HMI tags "03.PumpControl"
   "Stop" : Bool AT %M0.1, T100ms
   "Lo" : Bool AT %M0.2, T100ms
   "Start" : Bool AT %M0.0, T100ms
   "Hi" : Bool AT %M0.3, T100ms
   "P_1" : Bool AT %M0.4, T100ms
   "P_2" : Bool AT %M0.5, T100ms
   "P_3" : Bool AT %M0.6, T100ms
   "L" : Int AT %MW4, T100ms

text list "SystemTextList_ConfigErrorAlarmTextLibrary_1": 1 'NameService configuration error: Implicit deletion. Subelement instance @6%s@ must be deleted explicitly.'; 2 'NameService configuration error: Implicit deletion. Alias/Format/Unit instance @6%s@ must be deleted explicitly.'

text list "SystemTextList_ConfigErrorAlarmTextLibrary_2": 1 'EvDpManager::cleanupDeletedDatapoint - alert handler config is deleted implicitly for deleted datapoint, @3%s@'; 2 'EvDpManager::cleanupDeletedDatapoint - alert handler config is deleted implicitly but still has overrides, @3%s@'; 3 'EvDpManager::cleanupDeletedDatapoint - default value config is deleted implicitly for deleted datapoint, @3%s@'; 4 'EvDpManager::cleanupDeletedDatapoint - default value config is deleted implicitly but still has overrides, @3%s@'; 5 'EvDpManager::cleanupDeletedDatapoint - initial value config is deleted implicitly for deleted datapoint, @3%s@'; 6 'EvDpManager::cleanupDeletedDatapoint - initial value config is deleted implicitly but still has overrides, @3%s@'; 7 'EvDpManager::cleanupDeletedDatapoint - distribution config is deleted implicitly for deleted datapoint, @3%s@'; 8 'EvDpManager::cleanupDeletedDatapoint - distribution config is deleted implicitly but still has overrides, @3%s@'; 9 'EvDpManager::cleanupDeletedDatapoint - rangeCheck config is deleted implicitly for deleted datapoint, @3%s@'; 10 'EvDpManager::cleanupDeletedDatapoint - rangeCheck config is deleted implicitly but still has overrides, @3%s@'

text list "SystemTextList_ConfigErrorAlarmTextLibrary_3": 1 'The configured data point type was deleted, but a configured type is still defined for the node type: @3%s@.'; 2 'The configured data point node type was deleted in the data point type, but a configured type is still defined for the element: @3%s@.'

text list "SystemTextList_ConfigErrorAlarmTextLibrary_4": 2 'Cycles: @6%s@ does not exist'; 3 'Alarms: @6%s@ exists already'; 4 'Tags: Address @6%s@ was rejected'; 1 'Connections: @6%s@ does not exist'; 5 'Tags: Acquisition mode @6%s@ is not supported.'; 6 'Cycles: @6%s@ was deleted but associated tags exist.'; 7 'Connections: @6%s@ was deleted but associated tags exist.'; 8 'Tags: Tag @6%s@ was rejected.'; 9 'Tags: Tag @6%s@ has an invalid value.'; 0 'Connections: Connection to @6%s@ could not be established.'; 65638 'Connections: Connection to @6%s@ could not be established.'; 65639 'Connections: @6%s@ disconnected.'; 65640 'Connections: Connection to the HMI device @6%s@ is lost.'; 65641 'Connections: Connection to the PLC @6%s@ is lost.'; 65541 'Connections: Timeout while establishing the connection to @6%s@.'; 65542 'Connections: @6%s@ faulty.'; 65543 'Connections: Connection to the HMI device disconnected. Connection @5%s@ was changed.'; 65544 'Connections: Connection to the HMI device disconnected. Driver property was changed for connection @5%s@.'

text list "SystemTextList_ConfigErrorAlarmTextLibrary_5": 1 'Connections: Lifecycle monitoring cycle must be shorter than the response time.'; 2 'Connections: Cyclic services are configured but not supported by the target device.'; 3 'Connections: Change-controlled reading is configured but not supported by the target device.'; 4 'Tags: The address @6%s@ does not exist in the PLC.'; 5 'Tags: The default conversion type for the address @6%s@ could not be determined.'; 6 'Tags: Invalid conversion type'; 7 'Cycles: Invalid conversion type. Conversion is not supported at HmiCycle.'; 4096 'Connections: Version of the address @6%s@ is not supported.'; 4097 'Connections: PROFIBUS address is not supported.'; 4098 'Connections: Softbus address is not supported.'; 4099 'Connections: Address type @6%s@ is not supported.'; 4100 'Connections: Invalid connection name @6%s@. Access point is being ignored.'; 4101 'Connections: Routing is not supported. @6%s@ is not used.'; 4102 'Connections: Routing is not supported. @6%s@ is not used.'; 4103 'Connections: Invalid IP address @6%s@'; 4104 'Connections: Invalid Named Connection @6%s@. Valid format: >VMD</>connection<'; 4105 'Connections: Invalid Named Connection @6%s@. VMD connection name is too long. Only 24 characters are permitted.'; 4106 'Connections: Invalid Named Connection @6%s@. Connection name is too long. Only 32 characters are permitted.'; 4107 'Connections: Rack number @6%s@ is outside of the permitted range (0..7)'; 4108 'Connections: Invalid Named Connection @6%s@. Rack is ignored.'; 4109 'Connections: Slot number @6%s@ is outside of the permitted range (0..31)'; 4110 'Connections: Invalid Named Connection @6%s@. Slot is ignored.'; 4111 'Connection could not be established. Maximum number of available connections (@6%s@) has been exceeded.'; 4112 'Connection aborted. No sign of life in the last @4%s@ ms.'; 4113 'Connection could not be established - @4%s@'; 4114 'Connection could not be established. The address @6%s@ cannot be used.'; 4115 'Connection could not be established. Invalid address @6%s@'; 4116 'Connection could not be established - @4%s@'

text list "SystemTextList_ConfigErrorAlarmTextLibrary_6": 1 'Connection could not be established. Application instance certificate is not configured.'; 2 'Connection could not be established. Server has rejected the client certificate. OPC UA status code @4%s@.'; 3 'Connection could not be established. Internal problem in the certificate store. OPC UA status code @4%s@'; 4 'Connection could not be established. Application instance certificate could not be loaded. OPC UA status code @4%s@'; 5 'Connection could not be established. Server has not provided a certificate. @4%s@'; 6 'Connection could not be established. Validation of server certificate has failed. OPC UA status code @4%s@.'; 7 'Connection was closed. Error during alarm synchronization. OPC UA status code @4%s@.'; 8 'Connection was closed. Alarm/event subscription has failed. The number of operations on the server has been exceeded.'; 9 'Connection was closed. Alarm/event subscription has failed. The number of alarm/event subscriptions on the server has been exceeded.'; 10 'Connection could not be established. Server reports a license problem. OPC UA status code @4%s@.'; 11 'Connection could not be established. Maximum number of server sessions has been exceeded.'; 12 'Connection could not be established. Safety configuration is inconsistent. @4%s@'; 13 'Connection could not be established. The address @4%s@ cannot be used.'; 14 'Connection could not be established. OPC UA status code @4%s@'; 15 'Connection aborted. OPC UA server was stopped.'; 16 'Connection aborted. No sign of life in the last @4%s@ ms.'; 17 'Connection was closed. OPC UA server maintenance.'; 18 'Connection could not be established. Invalid configuration of the authentication mode - @4%s@'; 19 'Connection could not be established. User could not be authenticated. OPC UA status code @4%s@'; 20 'Connection could not be established. Server does not permit anonymous connection. OPC UA status code @4%s@'; 21 'Connection could not be established. Certificate problem: Error when writing the safety-relevant data to @4%s@.'; 22 'Connection could not be established. Certificate problem: Unexpected file in the folder @4%s@ cannot be removed.'; 23 'Connection could not be established. User could not be authenticated. No user or password configured.'; 24 'Connection could not be established. Unexpected length of the server certificate. @4%s@'; 25 'Connection could not be established. @4%s@ is empty.'; 26 'Connection could not be established. @4%s@ has an unexpected format.'; 27 'Connection could not be established. Server endpoints cannot be read. OPC UA status code @4%s@'; 28 'Connection could not be established. No server endpoints were found. @4%s@'; 29 'Connection could not be established. Application instance certificate could not be found.'; 30 'Connection could not be established. Unexpected format of the certificate @4%s@.'; 31 'Connection could not be established. Unexpected format of the certificate block list @4%s@.'; 32 'Connection could not be established. User could not be authenticated. An encryption detail is invalid. @4%s@'; 34 'Connection could not be established. - The configured non-transparent redundancy mode @4%s@ is not supported.'; 101 'Tags: Address @6%s@ does not exist on the server.'; 103 'Tags: Address @6%s@ cannot be accessed.'; 104 'Tags: Acquisition mode is not supported for address @6%s@.'; 201 'Alarms: Address @6%s@ does not exist on the server.'; 202 'Alarms: Address @6%s@ cannot be used. The specified range filter is not an OPC UA Event Notifier.'; 203 'Alarms: Address @6%s@ cannot be used. The specified range filter does not exist on the server.'; 204 'Alarms: Address @6%s@ cannot be used because it is not an OPC UA event type.'; 205 'Alarms: Address @6%s@ cannot be used because the OPC UA condition type is not supported.'; 206 'Alarms: Address @6%s@ cannot be used because the event type does not exist on the server.'; 207 'Alarms: Acquisition type cannot be used for address @6%s@.'; 301 'Address @6%s@ cannot be used because the version number is missing.'; 302 'Address @6%s@ cannot be used because the version number is invalid.'; 303 'Address @6%s@ cannot be used because the number of '$' delimiters is invalid.'; 304 'Address @6%s@ cannot be used because the address type is invalid.'; 305 'Unsupported version @6%s@ of the address'; 401 'Unexpected OPC UA server response: @6%s@'

text list "SystemTextList_ConfigErrorAlarmTextLibrary_7": 1 'Messages: Invalid condition string for the alarm view @6%s@.'; 2 'Messages: Invalid status tag and bit for the alarm view @6%s@.'; 3 'Messages: Invalid control tag and bit for the alarm view @6%s@.'

text list "SystemTextList_ConfigErrorAlarmTextLibrary_8": 1 'Logs: Implicit deletion. Logging tag instance @6%s@ should be deleted but there are overloaded elements.'

text list "SystemTextList_ConfigErrorAlarmTextLibrary_9": 2 'Restart of the runtime is required.'; 3 'The correct storage medium must be ejected and inserted again.'

text list "SystemTextList_ConfigErrorAlarmTextLibrary_10": 1 'CDS cache - Cache folder cannot be created or reached: @6%s@'; 2 'LOC cache - Cache folder cannot be created or reached: @6%s@'

text list "SystemTextList_ConfigErrorAlarmTextLibrary_11": 2 'and synchronization will start automatically. Shutting down either of them during synchronization will not cause data loss.'; 3 'and synchronization is scheduled for: @5%Y-%m-%d %H:%M:%S@. Shutting down either of the computers will not cause data loss.'

text list "SystemTextList_RuntimeCollaborationFailureReason_1": 0 'Unknown error (@3%s@)'; 1 'The system is not running or there is a network problem'; 2 'Runtime is not started on the target device.'; 3 'The System ID does not match the expected System ID (@3%s@)'; 4 'The Collaboration name does not match the expected Collaboration name '@3%s@''; 5 'Wrong or unknown certificate'; 6 'Revoked certificate'; 7 'The time difference is too big.'; 8 'No common supported message version'; 9 'System ID (@3%s@) already exists'; 10 'System name (@3%s@) already exists'; 11 'ID/Name in local configuration for Runtime Collaboration already exists'

text list "SystemTextList_RedundancyRecoveryFailureReason_1": 0 'Data recovery request temporarily rejected until own recovery request has been responded to.'; 1 'Data recovery request rejected. Online backup running.'; 2 'Data recovery request rejected. Connection to the Event Manager is not established.'; 3 'Data recovery request temporarily rejected until delta activation is complete.'; 4 'Data recovery request temporarily rejected until alarms and tags are retentive.'; 5 'Data recovery request rejected. The obligatory file config.level.es is missing on the computer.'; 6 'Data recovery request was canceled by the Event Manager.'; 7 'The data synchronization between the devices has failed.'

text list "SystemTextList_S7PlusAlarmTextListCollection_1": 4096 'Connections: Connection to the PLC @4%s@ is lost'; 4097 'Connections: Connection to the HMI device @4%s@ is lost'; 4098 'Connections: Maximum number of connections exceeded - @4%s@'; 4099 'Out of resources on PLC - @4%s@'; 4100 'Legitimation failed, invalid or missing password - @4%s@'; 4101 'Request to open the connection failed - @4%s@'; 4102 'Connections: Cannot connect to PLC - @4%s@'; 4103 'Request to open the connection could not be sent'; 4104 'General certificate error for PLC - @4%s@'; 4105 'PLC certificate expired for PLC - @4%s@'; 4106 'PLC certificate is revoked for PLC - @4%s@'; 4107 'PLC certificate is untrustworthy. Manual trust is possible for - @4%s@'; 4108 'PLC certificate is untrustworthy. Manual trust is not possible for - @4%s@'

text list "SystemTextList_AllenBradleyEIPAlarmTextListCollection_7": 4096 'Connection lost on PLC side - @5%s@'; 4097 'Connection lost on HMI side - @5%s@'; 4098 'Maximum number of connections exceeded - @5%s@'; 4099 'Out of resources on PLC - @5%s@'; 4100 'Legitimation failed, invalid or missing password - @5%s@'; 4101 'Open request failed - @5%s@'; 4102 'Cannot connect to PLC - @5%s@'; 4103 'Open request could not be sent'; 4104 'root certificate expired for - @5%s@'; 4105 'PLC certificate untrusted for - @5%s@'

text list "SystemTextList_AllenBradleyDF1AlarmTextListCollection_9": 4096 'Connections: Connection to the PLC @5%s@ is lost'; 4097 'Connections: Connection to the HMI device @5%s@ is lost'; 4098 'Connections: Maximum number of connections exceeded - @5%s@'; 4099 'Out of resources on PLC - @5%s@'; 4100 'Legitimation failed, invalid or missing password - @5%s@'; 4101 'Request to open the connection failed - @5%s@'; 4102 'Connections: Cannot connect to PLC - @5%s@'; 4103 'Request to open the connection could not be sent'; 4104 'General certificate error for PLC - @5%s@'; 4105 'PLC certificate expired for PLC - @5%s@'; 4106 'PLC certificate is revoked for PLC - @5%s@'; 4107 'PLC certificate is untrustworthy. Manual trust is possible for - @5%s@'; 4108 'PLC certificate is untrustworthy. Manual trust is not possible for - @5%s@'

text list "SystemTextList_OmronEIPAlarmTextListCollection_6": 4096 'Connection lost on PLC side - @5%s@'; 4097 'Connection lost on HMI side - @5%s@'; 4098 'Maximum number of connections exceeded - @5%s@'; 4099 'Out of resources on PLC - @5%s@'; 4100 'Legitimation failed, invalid or missing password - @5%s@'; 4101 'Open request failed - @5%s@'; 4102 'Cannot connect to PLC - @5%s@'; 4103 'Open request could not be sent'; 4104 'root certificate expired for - @5%s@'; 4105 'PLC certificate untrusted for - @5%s@'

text list "SystemTextList_StdModbusTCPAlarmTextListCollection_5": 4096 'Connections: Connection to the PLC @5%s@ is lost'; 4097 'Connections: Connection to the HMI device @5%s@ is lost'; 4098 'Connections: Maximum number of connections exceeded - @5%s@'; 4099 'Out of resources on PLC - @5%s@'; 4100 'Legitimation failed, invalid or missing password - @5%s@'; 4101 'Request to open the connection failed - @5%s@'; 4102 'Connections: Cannot connect to PLC - @5%s@'; 4103 'Request to open the connection could not be sent'; 4104 'General certificate error for PLC - @5%s@'; 4105 'PLC certificate expired for PLC - @5%s@'; 4106 'PLC certificate is revoked for PLC - @5%s@'; 4107 'PLC certificate is untrustworthy. Manual trust is possible for - @5%s@'; 4108 'PLC certificate is untrustworthy. Manual trust is not possible for - @5%s@'

text list "SystemTextList_MitsubishiMCAlarmTextListCollection_4": 4096 'Connection lost on PLC side - @5%s@'; 4097 'Connection lost on HMI side - @5%s@'; 4098 'Maximum number of connections exceeded - @5%s@'; 4099 'Out of resources on PLC - @5%s@'; 4100 'Legitimation failed, invalid or missing password - @5%s@'; 4101 'Open request failed - @5%s@'; 4102 'Cannot connect to PLC - @5%s@'; 4103 'Open request could not be sent'; 4104 'root certificate expired for - @5%s@'; 4105 'PLC certificate untrusted for - @5%s@'

text list "SystemTextList_MitsubishiiQAlarmTextListCollection_3": 4096 'Connection lost on PLC side - @5%s@'; 4097 'Connection lost on HMI side - @5%s@'; 4098 'Maximum number of connections exceeded - @5%s@'; 4099 'Out of resources on PLC - @5%s@'; 4100 'Legitimation failed, invalid or missing password - @5%s@'; 4101 'Open request failed - @5%s@'; 4102 'Cannot connect to PLC - @5%s@'; 4103 'Open request could not be sent'; 4104 'root certificate expired for - @5%s@'; 4105 'PLC certificate untrusted for - @5%s@'

text list "SystemTextList_StdModbusRTUAlarmTextListCollection_8": 4096 'Connections: Connection to the PLC @5%s@ is lost'; 4097 'Connections: Connection to the HMI device @5%s@ is lost'; 4098 'Connections: Maximum number of connections exceeded - @5%s@'; 4099 'Out of resources on PLC - @5%s@'; 4100 'Legitimation failed, invalid or missing password - @5%s@'; 4101 'Request to open the connection failed - @5%s@'; 4102 'Connections: Cannot connect to PLC - @5%s@'; 4103 'Request to open the connection could not be sent'; 4104 'General certificate error for PLC - @5%s@'; 4105 'PLC certificate expired for PLC - @5%s@'; 4106 'PLC certificate is revoked for PLC - @5%s@'; 4107 'PLC certificate is untrustworthy. Manual trust is possible for - @5%s@'; 4108 'PLC certificate is untrustworthy. Manual trust is not possible for - @5%s@'

text list "SystemTextList_LogoAlarmTextListCollection_10": 4096 'Connections: Connection to the PLC @5%s@ is lost'; 4097 'Connections: Connection to the HMI device @5%s@ is lost'; 4098 'Connections: Maximum number of connections exceeded - @5%s@'; 4099 'Out of resources on PLC - @5%s@'; 4100 'Legitimation failed, invalid or missing password - @5%s@'; 4101 'Request to open the connection failed - @5%s@'; 4102 'Connections: Cannot connect to PLC - @5%s@'; 4103 'Request to open the connection could not be sent'; 4104 'General certificate error for PLC - @5%s@'; 4105 'PLC certificate expired for PLC - @5%s@'; 4106 'PLC certificate is revoked for PLC - @5%s@'; 4107 'PLC certificate is untrustworthy. Manual trust is possible for - @5%s@'; 4108 'PLC certificate is untrustworthy. Manual trust is not possible for - @5%s@'

graphic list "Switch": 0 'rotary-switches-open'; 1 'rotary-switches-close'

graphic list "Light": 0 'light_green_off'; 1 'light_green_on'

graphic list "Agitator": 0 'agitator_1'; 1 'agitator_2'; 2 'agitator_3'; 3 'agitator_4'
*)

(* ===== HMI "HiddenHmiRTDeviceFaceplateTypes" =====

HMI tags "0daced1d-1c12-4c0f-a1c7-efedc7fbd37d"
   "Data" : f64981b7-23c1-4b9c-90a3-7c9aa74d9c52, internal
*)

(* ===== HMI "HiddenHmiRTDeviceFaceplateTypes" =====

HMI tags "0daced1d-1c12-4c0f-a1c7-efedc7fbd37d"
   "Data" : f64981b7-23c1-4b9c-90a3-7c9aa74d9c52, internal
*)

(* ===== HMI "HMI_RT_4" =====
connection "UA_Connection_1": SCADA_OPC, ILRT_OPC_UA
connection "S7_Connection_1": ETHERNET, ILRT_S7_1500_OMS

HMI tags "01.HeaterONOFFCtrl"
   "Temp_SP" : Float AT ns=http://www.siemens.com/simatic-s7-opcua;s="ON_OFF_Ctrl_1"."SP", T100ms
   "Temp" : Float AT ns=http://www.siemens.com/simatic-s7-opcua;s="ON_OFF_Ctrl_1"."T", T100ms
   "Enable" : Boolean AT ns=http://www.siemens.com/simatic-s7-opcua;s="ON_OFF_Ctrl_1"."Enable", T100ms
   "Ready" : Boolean AT ns=http://www.siemens.com/simatic-s7-opcua;s="HeaterSim_1"."Ready", T100ms
   "Fault" : Boolean AT ns=http://www.siemens.com/simatic-s7-opcua;s="HeaterSim_1"."Fault", T100ms

HMI tags "02.MotorDOLCtrl"
   "Theta" : Float AT ns=http://www.siemens.com/simatic-s7-opcua;s="MotorSim_1"."Theta", T100ms
   "Omega" : Real AT %DB4.DBD8, T100ms
   "EnableCtrl" : Boolean AT ns=http://www.siemens.com/simatic-s7-opcua;s="DOL_Ctrl_1"."Enable", T100ms
   "i_set" : Float AT ns=http://www.siemens.com/simatic-s7-opcua;s="DOL_Ctrl_1"."i_set", T100ms
   "RunCmd" : Boolean AT ns=http://www.siemens.com/simatic-s7-opcua;s="DOL_Ctrl_1"."RunCmd", T100ms
   "MotorFault" : Boolean AT ns=http://www.siemens.com/simatic-s7-opcua;s="MotorSim_1"."Fault", T100ms
   "MotorReady" : Boolean AT ns=http://www.siemens.com/simatic-s7-opcua;s="MotorSim_1"."Ready", T100ms

HMI tags "03.HeaterPIDCtrl"
   "Temperature_SP" : Real AT %DB6.DBD2, T100ms
   "Temperature" : Real AT %DB7.DBD8, T100ms
   "EnableHeaterCtrl" : Bool AT %DB6.DBX0.0, T100ms
   "HeaterReady" : Bool AT %DB7.DBX12.0, T100ms
   "Kp" : Real AT %DB6.DBD12, T100ms
   "Ki" : Real AT %DB6.DBD16, T100ms
   "Kd" : Real AT %DB6.DBD20, T100ms
   "u" : Real AT %DB6.DBD32, T100ms

HMI tags "04.MotorPIDCtrl"
   "Omega_SP_Motor" : Real AT %DB10.DBD2, T100ms
   "EnablePID_Motor" : Bool AT %DB10.DBX0.0, T100ms
   "RunCmd_Motor" : Bool AT %DB9.DBX0.1, T100ms
   "Ready_Motor" : Bool AT %DB8.DBX16.0, T100ms
   "Omega_Motor" : Real AT %DB10.DBD6, T100ms
   "Kd_Motor" : Real AT %DB10.DBD10, T100ms
   "Ki_Motor" : Real AT %DB10.DBD16, T100ms
   "Kp_Motor" : Real AT %DB10.DBD20, T100ms
   "u_Motor" : Real AT %DB10.DBD32, T100ms

text list "SystemTextList_ConfigErrorAlarmTextLibrary_1": 1 'NameService configuration error: Implicit deletion. Subelement instance @6%s@ must be deleted explicitly.'; 2 'NameService configuration error: Implicit deletion. Alias/Format/Unit instance @6%s@ must be deleted explicitly.'

text list "SystemTextList_ConfigErrorAlarmTextLibrary_2": 1 'EvDpManager::cleanupDeletedDatapoint - alert handler config is deleted implicitly for deleted datapoint, @3%s@'; 2 'EvDpManager::cleanupDeletedDatapoint - alert handler config is deleted implicitly but still has overrides, @3%s@'; 3 'EvDpManager::cleanupDeletedDatapoint - default value config is deleted implicitly for deleted datapoint, @3%s@'; 4 'EvDpManager::cleanupDeletedDatapoint - default value config is deleted implicitly but still has overrides, @3%s@'; 5 'EvDpManager::cleanupDeletedDatapoint - initial value config is deleted implicitly for deleted datapoint, @3%s@'; 6 'EvDpManager::cleanupDeletedDatapoint - initial value config is deleted implicitly but still has overrides, @3%s@'; 7 'EvDpManager::cleanupDeletedDatapoint - distribution config is deleted implicitly for deleted datapoint, @3%s@'; 8 'EvDpManager::cleanupDeletedDatapoint - distribution config is deleted implicitly but still has overrides, @3%s@'; 9 'EvDpManager::cleanupDeletedDatapoint - rangeCheck config is deleted implicitly for deleted datapoint, @3%s@'; 10 'EvDpManager::cleanupDeletedDatapoint - rangeCheck config is deleted implicitly but still has overrides, @3%s@'

text list "SystemTextList_ConfigErrorAlarmTextLibrary_3": 1 'The configured data point type was deleted, but a configured type is still defined for the node type: @3%s@.'; 2 'The configured data point node type was deleted in the data point type, but a configured type is still defined for the element: @3%s@.'

text list "SystemTextList_ConfigErrorAlarmTextLibrary_4": 2 'Cycles: @6%s@ does not exist'; 3 'Alarms: @6%s@ exists already'; 4 'Tags: Address @6%s@ was rejected'; 1 'Connections: @6%s@ does not exist'; 5 'Tags: Acquisition mode @6%s@ is not supported.'; 6 'Cycles: @6%s@ was deleted but associated tags exist.'; 7 'Connections: @6%s@ was deleted but associated tags exist.'; 8 'Tags: Tag @6%s@ was rejected.'; 9 'Tags: Tag @6%s@ has an invalid value.'; 0 'Connections: Connection to @6%s@ could not be established.'; 65638 'Connections: Connection to @6%s@ could not be established.'; 65639 'Connections: @6%s@ disconnected.'; 65640 'Connections: Connection to the HMI device @6%s@ is lost.'; 65641 'Connections: Connection to the PLC @6%s@ is lost.'; 65541 'Connections: Timeout while establishing the connection to @6%s@.'; 65542 'Connections: @6%s@ faulty.'; 65543 'Connections: Connection to the HMI device disconnected. Connection @5%s@ was changed.'; 65544 'Connections: Connection to the HMI device disconnected. Driver property was changed for connection @5%s@.'

text list "SystemTextList_ConfigErrorAlarmTextLibrary_5": 1 'Connections: Lifecycle monitoring cycle must be shorter than the response time.'; 2 'Connections: Cyclic services are configured but not supported by the target device.'; 3 'Connections: Change-controlled reading is configured but not supported by the target device.'; 4 'Tags: The address @6%s@ does not exist in the PLC.'; 5 'Tags: The default conversion type for the address @6%s@ could not be determined.'; 6 'Tags: Invalid conversion type'; 7 'Cycles: Invalid conversion type. Conversion is not supported at HmiCycle.'; 4096 'Connections: Version of the address @6%s@ is not supported.'; 4097 'Connections: PROFIBUS address is not supported.'; 4098 'Connections: Softbus address is not supported.'; 4099 'Connections: Address type @6%s@ is not supported.'; 4100 'Connections: Invalid connection name @6%s@. Access point is being ignored.'; 4101 'Connections: Routing is not supported. @6%s@ is not used.'; 4102 'Connections: Routing is not supported. @6%s@ is not used.'; 4103 'Connections: Invalid IP address @6%s@'; 4104 'Connections: Invalid Named Connection @6%s@. Valid format: >VMD</>connection<'; 4105 'Connections: Invalid Named Connection @6%s@. VMD connection name is too long. Only 24 characters are permitted.'; 4106 'Connections: Invalid Named Connection @6%s@. Connection name is too long. Only 32 characters are permitted.'; 4107 'Connections: Rack number @6%s@ is outside of the permitted range (0..7)'; 4108 'Connections: Invalid Named Connection @6%s@. Rack is ignored.'; 4109 'Connections: Slot number @6%s@ is outside of the permitted range (0..31)'; 4110 'Connections: Invalid Named Connection @6%s@. Slot is ignored.'; 4111 'Connection could not be established. Maximum number of available connections (@6%s@) has been exceeded.'; 4112 'Connection aborted. No sign of life in the last @4%s@ ms.'; 4113 'Connection could not be established - @4%s@'; 4114 'Connection could not be established. The address @6%s@ cannot be used.'; 4115 'Connection could not be established. Invalid address @6%s@'; 4116 'Connection could not be established - @4%s@'

text list "SystemTextList_ConfigErrorAlarmTextLibrary_6": 1 'Connection could not be established. Application instance certificate is not configured.'; 2 'Connection could not be established. Server has rejected the client certificate. OPC UA status code @4%s@.'; 3 'Connection could not be established. Internal problem in the certificate store. OPC UA status code @4%s@'; 4 'Connection could not be established. Application instance certificate could not be loaded. OPC UA status code @4%s@'; 5 'Connection could not be established. Server has not provided a certificate. @4%s@'; 6 'Connection could not be established. Validation of server certificate has failed. OPC UA status code @4%s@.'; 7 'Connection was closed. Error during alarm synchronization. OPC UA status code @4%s@.'; 8 'Connection was closed. Alarm/event subscription has failed. The number of operations on the server has been exceeded.'; 9 'Connection was closed. Alarm/event subscription has failed. The number of alarm/event subscriptions on the server has been exceeded.'; 10 'Connection could not be established. Server reports a license problem. OPC UA status code @4%s@.'; 11 'Connection could not be established. Maximum number of server sessions has been exceeded.'; 12 'Connection could not be established. Safety configuration is inconsistent. @4%s@'; 13 'Connection could not be established. The address @4%s@ cannot be used.'; 14 'Connection could not be established. OPC UA status code @4%s@'; 15 'Connection aborted. OPC UA server was stopped.'; 16 'Connection aborted. No sign of life in the last @4%s@ ms.'; 17 'Connection was closed. OPC UA server maintenance.'; 18 'Connection could not be established. Invalid configuration of the authentication mode - @4%s@'; 19 'Connection could not be established. User could not be authenticated. OPC UA status code @4%s@'; 20 'Connection could not be established. Server does not permit anonymous connection. OPC UA status code @4%s@'; 21 'Connection could not be established. Certificate problem: Error when writing the safety-relevant data to @4%s@.'; 22 'Connection could not be established. Certificate problem: Unexpected file in the folder @4%s@ cannot be removed.'; 23 'Connection could not be established. User could not be authenticated. No user or password configured.'; 24 'Connection could not be established. Unexpected length of the server certificate. @4%s@'; 25 'Connection could not be established. @4%s@ is empty.'; 26 'Connection could not be established. @4%s@ has an unexpected format.'; 27 'Connection could not be established. Server endpoints cannot be read. OPC UA status code @4%s@'; 28 'Connection could not be established. No server endpoints were found. @4%s@'; 29 'Connection could not be established. Application instance certificate could not be found.'; 30 'Connection could not be established. Unexpected format of the certificate @4%s@.'; 31 'Connection could not be established. Unexpected format of the certificate block list @4%s@.'; 32 'Connection could not be established. User could not be authenticated. An encryption detail is invalid. @4%s@'; 34 'Connection could not be established. - The configured non-transparent redundancy mode @4%s@ is not supported.'; 101 'Tags: Address @6%s@ does not exist on the server.'; 103 'Tags: Address @6%s@ cannot be accessed.'; 104 'Tags: Acquisition mode is not supported for address @6%s@.'; 201 'Alarms: Address @6%s@ does not exist on the server.'; 202 'Alarms: Address @6%s@ cannot be used. The specified range filter is not an OPC UA Event Notifier.'; 203 'Alarms: Address @6%s@ cannot be used. The specified range filter does not exist on the server.'; 204 'Alarms: Address @6%s@ cannot be used because it is not an OPC UA event type.'; 205 'Alarms: Address @6%s@ cannot be used because the OPC UA condition type is not supported.'; 206 'Alarms: Address @6%s@ cannot be used because the event type does not exist on the server.'; 207 'Alarms: Acquisition type cannot be used for address @6%s@.'; 301 'Address @6%s@ cannot be used because the version number is missing.'; 302 'Address @6%s@ cannot be used because the version number is invalid.'; 303 'Address @6%s@ cannot be used because the number of '$' delimiters is invalid.'; 304 'Address @6%s@ cannot be used because the address type is invalid.'; 305 'Unsupported version @6%s@ of the address'; 401 'Unexpected OPC UA server response: @6%s@'

text list "SystemTextList_ConfigErrorAlarmTextLibrary_7": 1 'Messages: Invalid condition string for the alarm view @6%s@.'; 2 'Messages: Invalid status tag and bit for the alarm view @6%s@.'; 3 'Messages: Invalid control tag and bit for the alarm view @6%s@.'

text list "SystemTextList_ConfigErrorAlarmTextLibrary_8": 1 'Logs: Implicit deletion. Logging tag instance @6%s@ should be deleted but there are overloaded elements.'

text list "SystemTextList_ConfigErrorAlarmTextLibrary_9": 2 'Restart of the runtime is required.'; 3 'The correct storage medium must be ejected and inserted again.'

text list "SystemTextList_ConfigErrorAlarmTextLibrary_10": 1 'CDS cache - Cache folder cannot be created or reached: @6%s@'; 2 'LOC cache - Cache folder cannot be created or reached: @6%s@'

text list "SystemTextList_ConfigErrorAlarmTextLibrary_11": 2 'and synchronization will start automatically. Shutting down either of them during synchronization will not cause data loss.'; 3 'and synchronization is scheduled for: @5%Y-%m-%d %H:%M:%S@. Shutting down either of the computers will not cause data loss.'

text list "SystemTextList_RuntimeCollaborationFailureReason_1": 0 'Unknown error (@3%s@)'; 1 'The system is not running or there is a network problem'; 2 'Runtime is not started on the target device.'; 3 'The System ID does not match the expected System ID (@3%s@)'; 4 'The Collaboration name does not match the expected Collaboration name '@3%s@''; 5 'Wrong or unknown certificate'; 6 'Revoked certificate'; 7 'The time difference is too big.'; 8 'No common supported message version'; 9 'System ID (@3%s@) already exists'; 10 'System name (@3%s@) already exists'; 11 'ID/Name in local configuration for Runtime Collaboration already exists'

text list "SystemTextList_RedundancyRecoveryFailureReason_1": 0 'Data recovery request temporarily rejected until own recovery request has been responded to.'; 1 'Data recovery request rejected. Online backup running.'; 2 'Data recovery request rejected. Connection to the Event Manager is not established.'; 3 'Data recovery request temporarily rejected until delta activation is complete.'; 4 'Data recovery request temporarily rejected until alarms and tags are retentive.'; 5 'Data recovery request rejected. The obligatory file config.level.es is missing on the computer.'; 6 'Data recovery request was canceled by the Event Manager.'; 7 'The data synchronization between the devices has failed.'

text list "SystemTextList_S7PlusAlarmTextListCollection_1": 4096 'Connections: Connection to the PLC @4%s@ is lost'; 4097 'Connections: Connection to the HMI device @4%s@ is lost'; 4098 'Connections: Maximum number of connections exceeded - @4%s@'; 4099 'Out of resources on PLC - @4%s@'; 4100 'Legitimation failed, invalid or missing password - @4%s@'; 4101 'Request to open the connection failed - @4%s@'; 4102 'Connections: Cannot connect to PLC - @4%s@'; 4103 'Request to open the connection could not be sent'; 4104 'General certificate error for PLC - @4%s@'; 4105 'PLC certificate expired for PLC - @4%s@'; 4106 'PLC certificate is revoked for PLC - @4%s@'; 4107 'PLC certificate is untrustworthy. Manual trust is possible for - @4%s@'; 4108 'PLC certificate is untrustworthy. Manual trust is not possible for - @4%s@'

text list "SystemTextList_AllenBradleyEIPAlarmTextListCollection_7": 4096 'Connection lost on PLC side - @5%s@'; 4097 'Connection lost on HMI side - @5%s@'; 4098 'Maximum number of connections exceeded - @5%s@'; 4099 'Out of resources on PLC - @5%s@'; 4100 'Legitimation failed, invalid or missing password - @5%s@'; 4101 'Open request failed - @5%s@'; 4102 'Cannot connect to PLC - @5%s@'; 4103 'Open request could not be sent'; 4104 'root certificate expired for - @5%s@'; 4105 'PLC certificate untrusted for - @5%s@'

text list "SystemTextList_AllenBradleyDF1AlarmTextListCollection_9": 4096 'Connections: Connection to the PLC @5%s@ is lost'; 4097 'Connections: Connection to the HMI device @5%s@ is lost'; 4098 'Connections: Maximum number of connections exceeded - @5%s@'; 4099 'Out of resources on PLC - @5%s@'; 4100 'Legitimation failed, invalid or missing password - @5%s@'; 4101 'Request to open the connection failed - @5%s@'; 4102 'Connections: Cannot connect to PLC - @5%s@'; 4103 'Request to open the connection could not be sent'; 4104 'General certificate error for PLC - @5%s@'; 4105 'PLC certificate expired for PLC - @5%s@'; 4106 'PLC certificate is revoked for PLC - @5%s@'; 4107 'PLC certificate is untrustworthy. Manual trust is possible for - @5%s@'; 4108 'PLC certificate is untrustworthy. Manual trust is not possible for - @5%s@'

text list "SystemTextList_OmronEIPAlarmTextListCollection_6": 4096 'Connection lost on PLC side - @5%s@'; 4097 'Connection lost on HMI side - @5%s@'; 4098 'Maximum number of connections exceeded - @5%s@'; 4099 'Out of resources on PLC - @5%s@'; 4100 'Legitimation failed, invalid or missing password - @5%s@'; 4101 'Open request failed - @5%s@'; 4102 'Cannot connect to PLC - @5%s@'; 4103 'Open request could not be sent'; 4104 'root certificate expired for - @5%s@'; 4105 'PLC certificate untrusted for - @5%s@'

text list "SystemTextList_StdModbusTCPAlarmTextListCollection_5": 4096 'Connections: Connection to the PLC @5%s@ is lost'; 4097 'Connections: Connection to the HMI device @5%s@ is lost'; 4098 'Connections: Maximum number of connections exceeded - @5%s@'; 4099 'Out of resources on PLC - @5%s@'; 4100 'Legitimation failed, invalid or missing password - @5%s@'; 4101 'Request to open the connection failed - @5%s@'; 4102 'Connections: Cannot connect to PLC - @5%s@'; 4103 'Request to open the connection could not be sent'; 4104 'General certificate error for PLC - @5%s@'; 4105 'PLC certificate expired for PLC - @5%s@'; 4106 'PLC certificate is revoked for PLC - @5%s@'; 4107 'PLC certificate is untrustworthy. Manual trust is possible for - @5%s@'; 4108 'PLC certificate is untrustworthy. Manual trust is not possible for - @5%s@'

text list "SystemTextList_MitsubishiMCAlarmTextListCollection_4": 4096 'Connection lost on PLC side - @5%s@'; 4097 'Connection lost on HMI side - @5%s@'; 4098 'Maximum number of connections exceeded - @5%s@'; 4099 'Out of resources on PLC - @5%s@'; 4100 'Legitimation failed, invalid or missing password - @5%s@'; 4101 'Open request failed - @5%s@'; 4102 'Cannot connect to PLC - @5%s@'; 4103 'Open request could not be sent'; 4104 'root certificate expired for - @5%s@'; 4105 'PLC certificate untrusted for - @5%s@'

text list "SystemTextList_MitsubishiiQAlarmTextListCollection_3": 4096 'Connection lost on PLC side - @5%s@'; 4097 'Connection lost on HMI side - @5%s@'; 4098 'Maximum number of connections exceeded - @5%s@'; 4099 'Out of resources on PLC - @5%s@'; 4100 'Legitimation failed, invalid or missing password - @5%s@'; 4101 'Open request failed - @5%s@'; 4102 'Cannot connect to PLC - @5%s@'; 4103 'Open request could not be sent'; 4104 'root certificate expired for - @5%s@'; 4105 'PLC certificate untrusted for - @5%s@'

text list "SystemTextList_StdModbusRTUAlarmTextListCollection_8": 4096 'Connections: Connection to the PLC @5%s@ is lost'; 4097 'Connections: Connection to the HMI device @5%s@ is lost'; 4098 'Connections: Maximum number of connections exceeded - @5%s@'; 4099 'Out of resources on PLC - @5%s@'; 4100 'Legitimation failed, invalid or missing password - @5%s@'; 4101 'Request to open the connection failed - @5%s@'; 4102 'Connections: Cannot connect to PLC - @5%s@'; 4103 'Request to open the connection could not be sent'; 4104 'General certificate error for PLC - @5%s@'; 4105 'PLC certificate expired for PLC - @5%s@'; 4106 'PLC certificate is revoked for PLC - @5%s@'; 4107 'PLC certificate is untrustworthy. Manual trust is possible for - @5%s@'; 4108 'PLC certificate is untrustworthy. Manual trust is not possible for - @5%s@'

text list "SystemTextList_LogoAlarmTextListCollection_10": 4096 'Connections: Connection to the PLC @5%s@ is lost'; 4097 'Connections: Connection to the HMI device @5%s@ is lost'; 4098 'Connections: Maximum number of connections exceeded - @5%s@'; 4099 'Out of resources on PLC - @5%s@'; 4100 'Legitimation failed, invalid or missing password - @5%s@'; 4101 'Request to open the connection failed - @5%s@'; 4102 'Connections: Cannot connect to PLC - @5%s@'; 4103 'Request to open the connection could not be sent'; 4104 'General certificate error for PLC - @5%s@'; 4105 'PLC certificate expired for PLC - @5%s@'; 4106 'PLC certificate is revoked for PLC - @5%s@'; 4107 'PLC certificate is untrustworthy. Manual trust is possible for - @5%s@'; 4108 'PLC certificate is untrustworthy. Manual trust is not possible for - @5%s@'

graphic list "Switch": 0 'rotary-switches-open'; 1 'rotary-switches-close'

graphic list "Light": 0 'light_green_off'; 1 'light_green_on'

graphic list "Agitator": 0 'agitator_1'; 1 'agitator_2'; 2 'agitator_3'; 3 'agitator_4'
*)

(* ===== HMI "HiddenHmiRTDeviceFaceplateTypes" =====

HMI tags "8162c4aa-2830-459f-8ab4-a2eb131a0399"
   "V" : Real, internal
   "Vab" : Real, internal
   "Vbc" : Real, internal
   "Vca" : Real, internal
   "I" : Real, internal
   "Ia" : Real, internal
   "Ib" : Real, internal
   "Ic" : Real, internal
   "P" : Real, internal
   "Q" : Real, internal
   "PF" : Real, internal
   "E" : Real, internal
   "ID" : Real, internal
   "CB_1" : Bool, internal
   "CB_2" : Bool, internal
   "CB_3" : Bool, internal
*)

(* ===== HMI "Energy Management" =====
connection "Device_01": ETHERNET, UnifiedStdModbusTCP
connection "Device_02": ETHERNET, UnifiedStdModbusTCP
connection "Device_03": ETHERNET, UnifiedStdModbusTCP
connection "Device_04": ETHERNET, UnifiedStdModbusTCP
connection "Device_05": ETHERNET, UnifiedStdModbusTCP
connection "Device_06": ETHERNET, UnifiedStdModbusTCP
connection "Device_07": ETHERNET, UnifiedStdModbusTCP
connection "Device_08": ETHERNET, UnifiedStdModbusTCP
connection "Device_09": ETHERNET, UnifiedStdModbusTCP
connection "Device_10": ETHERNET, UnifiedStdModbusTCP
connection "Device_11": ETHERNET, UnifiedStdModbusTCP
connection "Device_12": ETHERNET, UnifiedStdModbusTCP
connection "Device_13": ETHERNET, UnifiedStdModbusTCP
connection "Device_14": ETHERNET, UnifiedStdModbusTCP
connection "Device_15": ETHERNET, UnifiedStdModbusTCP
connection "Device_16": ETHERNET, UnifiedStdModbusTCP
connection "Device_17": ETHERNET, UnifiedStdModbusTCP
connection "Device_18": ETHERNET, UnifiedStdModbusTCP
connection "Device_19": ETHERNET, UnifiedStdModbusTCP
connection "Device_20": ETHERNET, UnifiedStdModbusTCP

HMI tags "Tags"
   "PM_1_V" : Float AT 4x400001, T100ms
   "PM_1_Vab" : Float AT 4x400003, T100ms
   "PM_1_Vbc" : Float AT 4x400005, T100ms
   "PM_1_Vca" : Float AT 4x400007, T100ms
   "PM_1_I" : Float AT 4x400009, T100ms
   "PM_1_Ia" : Float AT 4x400011, T100ms
   "PM_1_Ib" : Float AT 4x400013, T100ms
   "PM_1_Ic" : Float AT 4x400015, T100ms
   "PM_1_P" : Float AT 4x400017, T100ms
   "PM_1_Q" : Float AT 4x400019, T100ms
   "PM_1_PF" : Float AT 4x400021, T100ms
   "PM_1_E" : Float AT 4x400023, T100ms
   "PM_1_CB_1" : Bit AT 0x1, T100ms
   "PM_1_CB_2" : Bit AT 0x2, T100ms
   "PM_1_CB_3" : Bit AT 0x3, T100ms
   "PM_1_ID" : Float AT 4x400025, T100ms
   "PM_2_V" : Float AT 4x400001, T100ms
   "PM_2_Vab" : Float AT 4x400003, T100ms
   "PM_2_Vbc" : Float AT 4x400005, T100ms
   "PM_2_Vca" : Float AT 4x400007, T100ms
   "PM_2_I" : Float AT 4x400009, T100ms
   "PM_2_Ia" : Float AT 4x400011, T100ms
   "PM_2_Ib" : Float AT 4x400013, T100ms
   "PM_2_Ic" : Float AT 4x400015, T100ms
   "PM_2_P" : Float AT 4x400017, T100ms
   "PM_2_Q" : Float AT 4x400019, T100ms
   "PM_2_PF" : Float AT 4x400021, T100ms
   "PM_2_E" : Float AT 4x400023, T100ms
   "PM_2_CB_1" : Bit AT 0x1, T100ms
   "PM_2_CB_2" : Bit AT 0x2, T100ms
   "PM_2_CB_3" : Bit AT 0x3, T100ms
   "PM_2_ID" : Float AT 4x400025, T100ms
   "PM_3_V" : Float AT 4x400001, T100ms
   "PM_3_Vab" : Float AT 4x400003, T100ms
   "PM_3_Vbc" : Float AT 4x400005, T100ms
   "PM_3_Vca" : Float AT 4x400007, T100ms
   "PM_3_I" : Float AT 4x400009, T100ms
   "PM_3_Ia" : Float AT 4x400011, T100ms
   "PM_3_Ib" : Float AT 4x400013, T100ms
   "PM_3_Ic" : Float AT 4x400015, T100ms
   "PM_3_P" : Float AT 4x400017, T100ms
   "PM_3_Q" : Float AT 4x400019, T100ms
   "PM_3_PF" : Float AT 4x400021, T100ms
   "PM_3_E" : Float AT 4x400023, T100ms
   "PM_3_CB_1" : Bit AT 0x1, T100ms
   "PM_3_CB_2" : Bit AT 0x2, T100ms
   "PM_3_CB_3" : Bit AT 0x3, T100ms
   "PM_3_ID" : Float AT 4x400025, T100ms
   "PM_4_V" : Float AT 4x400001, T100ms
   "PM_4_Vab" : Float AT 4x400003, T100ms
   "PM_4_Vbc" : Float AT 4x400005, T100ms
   "PM_4_Vca" : Float AT 4x400007, T100ms
   "PM_4_I" : Float AT 4x400009, T100ms
   "PM_4_Ia" : Float AT 4x400011, T100ms
   "PM_4_Ib" : Float AT 4x400013, T100ms
   "PM_4_Ic" : Float AT 4x400015, T100ms
   "PM_4_P" : Float AT 4x400017, T100ms
   "PM_4_Q" : Float AT 4x400019, T100ms
   "PM_4_PF" : Float AT 4x400021, T100ms
   "PM_4_E" : Float AT 4x400023, T100ms
   "PM_4_CB_1" : Bit AT 0x1, T100ms
   "PM_4_CB_2" : Bit AT 0x2, T100ms
   "PM_4_CB_3" : Bit AT 0x3, T100ms
   "PM_4_ID" : Float AT 4x400025, T100ms
   "PM_5_V" : Float AT 4x400001, T100ms
   "PM_5_Vab" : Float AT 4x400003, T100ms
   "PM_5_Vbc" : Float AT 4x400005, T100ms
   "PM_5_Vca" : Float AT 4x400007, T100ms
   "PM_5_I" : Float AT 4x400009, T100ms
   "PM_5_Ia" : Float AT 4x400011, T100ms
   "PM_5_Ib" : Float AT 4x400013, T100ms
   "PM_5_Ic" : Float AT 4x400015, T100ms
   "PM_5_P" : Float AT 4x400017, T100ms
   "PM_5_Q" : Float AT 4x400019, T100ms
   "PM_5_PF" : Float AT 4x400021, T100ms
   "PM_5_E" : Float AT 4x400023, T100ms
   "PM_5_CB_1" : Bit AT 0x1, T100ms
   "PM_5_CB_2" : Bit AT 0x2, T100ms
   "PM_5_CB_3" : Bit AT 0x3, T100ms
   "PM_5_ID" : Float AT 4x400025, T100ms
   "PM_6_V" : Float AT 4x400001, T100ms
   "PM_6_Vab" : Float AT 4x400003, T100ms
   "PM_6_Vbc" : Float AT 4x400005, T100ms
   "PM_6_Vca" : Float AT 4x400007, T100ms
   "PM_6_I" : Float AT 4x400009, T100ms
   "PM_6_Ia" : Float AT 4x400011, T100ms
   "PM_6_Ib" : Float AT 4x400013, T100ms
   "PM_6_Ic" : Float AT 4x400015, T100ms
   "PM_6_P" : Float AT 4x400017, T100ms
   "PM_6_Q" : Float AT 4x400019, T100ms
   "PM_6_PF" : Float AT 4x400021, T100ms
   "PM_6_E" : Float AT 4x400023, T100ms
   "PM_6_CB_1" : Bit AT 0x1, T100ms
   "PM_6_CB_2" : Bit AT 0x2, T100ms
   "PM_6_CB_3" : Bit AT 0x3, T100ms
   "PM_6_ID" : Float AT 4x400025, T100ms
   "PM_7_V" : Float AT 4x400001, T100ms
   "PM_7_Vab" : Float AT 4x400003, T100ms
   "PM_7_Vbc" : Float AT 4x400005, T100ms
   "PM_7_Vca" : Float AT 4x400007, T100ms
   "PM_7_I" : Float AT 4x400009, T100ms
   "PM_7_Ia" : Float AT 4x400011, T100ms
   "PM_7_Ib" : Float AT 4x400013, T100ms
   "PM_7_Ic" : Float AT 4x400015, T100ms
   "PM_7_P" : Float AT 4x400017, T100ms
   "PM_7_Q" : Float AT 4x400019, T100ms
   "PM_7_PF" : Float AT 4x400021, T100ms
   "PM_7_E" : Float AT 4x400023, T100ms
   "PM_7_CB_1" : Bit AT 0x1, T100ms
   "PM_7_CB_2" : Bit AT 0x2, T100ms
   "PM_7_CB_3" : Bit AT 0x3, T100ms
   "PM_7_ID" : Float AT 4x400025, T100ms
   "PM_8_V" : Float AT 4x400001, T100ms
   "PM_8_Vab" : Float AT 4x400003, T100ms
   "PM_8_Vbc" : Float AT 4x400005, T100ms
   "PM_8_Vca" : Float AT 4x400007, T100ms
   "PM_8_I" : Float AT 4x400009, T100ms
   "PM_8_Ia" : Float AT 4x400011, T100ms
   "PM_8_Ib" : Float AT 4x400013, T100ms
   "PM_8_Ic" : Float AT 4x400015, T100ms
   "PM_8_P" : Float AT 4x400017, T100ms
   "PM_8_Q" : Float AT 4x400019, T100ms
   "PM_8_PF" : Float AT 4x400021, T100ms
   "PM_8_E" : Float AT 4x400023, T100ms
   "PM_8_CB_1" : Bit AT 0x1, T100ms
   "PM_8_CB_2" : Bit AT 0x2, T100ms
   "PM_8_CB_3" : Bit AT 0x3, T100ms
   "PM_8_ID" : Float AT 4x400025, T100ms
   "PM_9_V" : Float AT 4x400001, T100ms
   "PM_9_Vab" : Float AT 4x400003, T100ms
   "PM_9_Vbc" : Float AT 4x400005, T100ms
   "PM_9_Vca" : Float AT 4x400007, T100ms
   "PM_9_I" : Float AT 4x400009, T100ms
   "PM_9_Ia" : Float AT 4x400011, T100ms
   "PM_9_Ib" : Float AT 4x400013, T100ms
   "PM_9_Ic" : Float AT 4x400015, T100ms
   "PM_9_P" : Float AT 4x400017, T100ms
   "PM_9_Q" : Float AT 4x400019, T100ms
   "PM_9_PF" : Float AT 4x400021, T100ms
   "PM_9_E" : Float AT 4x400023, T100ms
   "PM_9_CB_1" : Bit AT 0x1, T100ms
   "PM_9_CB_2" : Bit AT 0x2, T100ms
   "PM_9_CB_3" : Bit AT 0x3, T100ms
   "PM_9_ID" : Float AT 4x400025, T100ms
   "PM_10_V" : Float AT 4x400001, T100ms
   "PM_10_Vab" : Float AT 4x400003, T100ms
   "PM_10_Vbc" : Float AT 4x400005, T100ms
   "PM_10_Vca" : Float AT 4x400007, T100ms
   "PM_10_I" : Float AT 4x400009, T100ms
   "PM_10_Ia" : Float AT 4x400011, T100ms
   "PM_10_Ib" : Float AT 4x400013, T100ms
   "PM_10_Ic" : Float AT 4x400015, T100ms
   "PM_10_P" : Float AT 4x400017, T100ms
   "PM_10_Q" : Float AT 4x400019, T100ms
   "PM_10_PF" : Float AT 4x400021, T100ms
   "PM_10_E" : Float AT 4x400023, T100ms
   "PM_10_CB_1" : Bit AT 0x1, T100ms
   "PM_10_CB_2" : Bit AT 0x2, T100ms
   "PM_10_CB_3" : Bit AT 0x3, T100ms
   "PM_10_ID" : Float AT 4x400025, T100ms
   "PM_11_V" : Float AT 4x400001, T100ms
   "PM_11_Vab" : Float AT 4x400003, T100ms
   "PM_11_Vbc" : Float AT 4x400005, T100ms
   "PM_11_Vca" : Float AT 4x400007, T100ms
   "PM_11_I" : Float AT 4x400009, T100ms
   "PM_11_Ia" : Float AT 4x400011, T100ms
   "PM_11_Ib" : Float AT 4x400013, T100ms
   "PM_11_Ic" : Float AT 4x400015, T100ms
   "PM_11_P" : Float AT 4x400017, T100ms
   "PM_11_Q" : Float AT 4x400019, T100ms
   "PM_11_PF" : Float AT 4x400021, T100ms
   "PM_11_E" : Float AT 4x400023, T100ms
   "PM_11_CB_1" : Bit AT 0x1, T100ms
   "PM_11_CB_2" : Bit AT 0x2, T100ms
   "PM_11_CB_3" : Bit AT 0x3, T100ms
   "PM_11_ID" : Float AT 4x400025, T100ms
   "PM_12_V" : Float AT 4x400001, T100ms
   "PM_12_Vab" : Float AT 4x400003, T100ms
   "PM_12_Vbc" : Float AT 4x400005, T100ms
   "PM_12_Vca" : Float AT 4x400007, T100ms
   "PM_12_I" : Float AT 4x400009, T100ms
   "PM_12_Ia" : Float AT 4x400011, T100ms
   "PM_12_Ib" : Float AT 4x400013, T100ms
   "PM_12_Ic" : Float AT 4x400015, T100ms
   "PM_12_P" : Float AT 4x400017, T100ms
   "PM_12_Q" : Float AT 4x400019, T100ms
   "PM_12_PF" : Float AT 4x400021, T100ms
   "PM_12_E" : Float AT 4x400023, T100ms
   "PM_12_CB_1" : Bit AT 0x1, T100ms
   "PM_12_CB_2" : Bit AT 0x2, T100ms
   "PM_12_CB_3" : Bit AT 0x3, T100ms
   "PM_12_ID" : Float AT 4x400025, T100ms
   "PM_13_V" : Float AT 4x400001, T100ms
   "PM_13_Vab" : Float AT 4x400003, T100ms
   "PM_13_Vbc" : Float AT 4x400005, T100ms
   "PM_13_Vca" : Float AT 4x400007, T100ms
   "PM_13_I" : Float AT 4x400009, T100ms
   "PM_13_Ia" : Float AT 4x400011, T100ms
   "PM_13_Ib" : Float AT 4x400013, T100ms
   "PM_13_Ic" : Float AT 4x400015, T100ms
   "PM_13_P" : Float AT 4x400017, T100ms
   "PM_13_Q" : Float AT 4x400019, T100ms
   "PM_13_PF" : Float AT 4x400021, T100ms
   "PM_13_E" : Float AT 4x400023, T100ms
   "PM_13_CB_1" : Bit AT 0x1, T100ms
   "PM_13_CB_2" : Bit AT 0x2, T100ms
   "PM_13_CB_3" : Bit AT 0x3, T100ms
   "PM_13_ID" : Float AT 4x400025, T100ms
   "PM_14_V" : Float AT 4x400001, T100ms
   "PM_14_Vab" : Float AT 4x400003, T100ms
   "PM_14_Vbc" : Float AT 4x400005, T100ms
   "PM_14_Vca" : Float AT 4x400007, T100ms
   "PM_14_I" : Float AT 4x400009, T100ms
   "PM_14_Ia" : Float AT 4x400011, T100ms
   "PM_14_Ib" : Float AT 4x400013, T100ms
   "PM_14_Ic" : Float AT 4x400015, T100ms
   "PM_14_P" : Float AT 4x400017, T100ms
   "PM_14_Q" : Float AT 4x400019, T100ms
   "PM_14_PF" : Float AT 4x400021, T100ms
   "PM_14_E" : Float AT 4x400023, T100ms
   "PM_14_CB_1" : Bit AT 0x1, T100ms
   "PM_14_CB_2" : Bit AT 0x2, T100ms
   "PM_14_CB_3" : Bit AT 0x3, T100ms
   "PM_14_ID" : Float AT 4x400025, T100ms
   "PM_15_V" : Float AT 4x400001, T100ms
   "PM_15_Vab" : Float AT 4x400003, T100ms
   "PM_15_Vbc" : Float AT 4x400005, T100ms
   "PM_15_Vca" : Float AT 4x400007, T100ms
   "PM_15_I" : Float AT 4x400009, T100ms
   "PM_15_Ia" : Float AT 4x400011, T100ms
   "PM_15_Ib" : Float AT 4x400013, T100ms
   "PM_15_Ic" : Float AT 4x400015, T100ms
   "PM_15_P" : Float AT 4x400017, T100ms
   "PM_15_Q" : Float AT 4x400019, T100ms
   "PM_15_PF" : Float AT 4x400021, T100ms
   "PM_15_E" : Float AT 4x400023, T100ms
   "PM_15_CB_1" : Bit AT 0x1, T100ms
   "PM_15_CB_2" : Bit AT 0x2, T100ms
   "PM_15_CB_3" : Bit AT 0x3, T100ms
   "PM_15_ID" : Float AT 4x400025, T100ms
   "PM_16_V" : Float AT 4x400001, T100ms
   "PM_16_Vab" : Float AT 4x400003, T100ms
   "PM_16_Vbc" : Float AT 4x400005, T100ms
   "PM_16_Vca" : Float AT 4x400007, T100ms
   "PM_16_I" : Float AT 4x400009, T100ms
   "PM_16_Ia" : Float AT 4x400011, T100ms
   "PM_16_Ib" : Float AT 4x400013, T100ms
   "PM_16_Ic" : Float AT 4x400015, T100ms
   "PM_16_P" : Float AT 4x400017, T100ms
   "PM_16_Q" : Float AT 4x400019, T100ms
   "PM_16_PF" : Float AT 4x400021, T100ms
   "PM_16_E" : Float AT 4x400023, T100ms
   "PM_16_CB_1" : Bit AT 0x1, T100ms
   "PM_16_CB_2" : Bit AT 0x2, T100ms
   "PM_16_CB_3" : Bit AT 0x3, T100ms
   "PM_16_ID" : Float AT 4x400025, T100ms
   "PM_17_V" : Float AT 4x400001, T100ms
   "PM_17_Vab" : Float AT 4x400003, T100ms
   "PM_17_Vbc" : Float AT 4x400005, T100ms
   "PM_17_Vca" : Float AT 4x400007, T100ms
   "PM_17_I" : Float AT 4x400009, T100ms
   "PM_17_Ia" : Float AT 4x400011, T100ms
   "PM_17_Ib" : Float AT 4x400013, T100ms
   "PM_17_Ic" : Float AT 4x400015, T100ms
   "PM_17_P" : Float AT 4x400017, T100ms
   "PM_17_Q" : Float AT 4x400019, T100ms
   "PM_17_PF" : Float AT 4x400021, T100ms
   "PM_17_E" : Float AT 4x400023, T100ms
   "PM_17_CB_1" : Bit AT 0x1, T100ms
   "PM_17_CB_2" : Bit AT 0x2, T100ms
   "PM_17_CB_3" : Bit AT 0x3, T100ms
   "PM_17_ID" : Float AT 4x400025, T100ms
   "PM_18_V" : Float AT 4x400001, T100ms
   "PM_18_Vab" : Float AT 4x400003, T100ms
   "PM_18_Vbc" : Float AT 4x400005, T100ms
   "PM_18_Vca" : Float AT 4x400007, T100ms
   "PM_18_I" : Float AT 4x400009, T100ms
   "PM_18_Ia" : Float AT 4x400011, T100ms
   "PM_18_Ib" : Float AT 4x400013, T100ms
   "PM_18_Ic" : Float AT 4x400015, T100ms
   "PM_18_P" : Float AT 4x400017, T100ms
   "PM_18_Q" : Float AT 4x400019, T100ms
   "PM_18_PF" : Float AT 4x400021, T100ms
   "PM_18_E" : Float AT 4x400023, T100ms
   "PM_18_CB_1" : Bit AT 0x1, T100ms
   "PM_18_CB_2" : Bit AT 0x2, T100ms
   "PM_18_CB_3" : Bit AT 0x3, T100ms
   "PM_18_ID" : Float AT 4x400025, T100ms
   "PM_19_V" : Float AT 4x400001, T100ms
   "PM_19_Vab" : Float AT 4x400003, T100ms
   "PM_19_Vbc" : Float AT 4x400005, T100ms
   "PM_19_Vca" : Float AT 4x400007, T100ms
   "PM_19_I" : Float AT 4x400009, T100ms
   "PM_19_Ia" : Float AT 4x400011, T100ms
   "PM_19_Ib" : Float AT 4x400013, T100ms
   "PM_19_Ic" : Float AT 4x400015, T100ms
   "PM_19_P" : Float AT 4x400017, T100ms
   "PM_19_Q" : Float AT 4x400019, T100ms
   "PM_19_PF" : Float AT 4x400021, T100ms
   "PM_19_E" : Float AT 4x400023, T100ms
   "PM_19_CB_1" : Bit AT 0x1, T100ms
   "PM_19_CB_2" : Bit AT 0x2, T100ms
   "PM_19_CB_3" : Bit AT 0x3, T100ms
   "PM_19_ID" : Float AT 4x400025, T100ms
   "PM_20_V" : Float AT 4x400001, T100ms
   "PM_20_Vab" : Float AT 4x400003, T100ms
   "PM_20_Vbc" : Float AT 4x400005, T100ms
   "PM_20_Vca" : Float AT 4x400007, T100ms
   "PM_20_I" : Float AT 4x400009, T100ms
   "PM_20_Ia" : Float AT 4x400011, T100ms
   "PM_20_Ib" : Float AT 4x400013, T100ms
   "PM_20_Ic" : Float AT 4x400015, T100ms
   "PM_20_P" : Float AT 4x400017, T100ms
   "PM_20_Q" : Float AT 4x400019, T100ms
   "PM_20_PF" : Float AT 4x400021, T100ms
   "PM_20_E" : Float AT 4x400023, T100ms
   "PM_20_CB_1" : Bit AT 0x1, T100ms
   "PM_20_CB_2" : Bit AT 0x2, T100ms
   "PM_20_CB_3" : Bit AT 0x3, T100ms
   "PM_20_ID" : Float AT 4x400025, T100ms

text list "SystemTextList_ConfigErrorAlarmTextLibrary_1": 1 'NameService configuration error: Implicit deletion. Subelement instance @6%s@ must be deleted explicitly.'; 2 'NameService configuration error: Implicit deletion. Alias/Format/Unit instance @6%s@ must be deleted explicitly.'

text list "SystemTextList_ConfigErrorAlarmTextLibrary_2": 1 'EvDpManager::cleanupDeletedDatapoint - alert handler config is deleted implicitly for deleted datapoint, @3%s@'; 2 'EvDpManager::cleanupDeletedDatapoint - alert handler config is deleted implicitly but still has overrides, @3%s@'; 3 'EvDpManager::cleanupDeletedDatapoint - default value config is deleted implicitly for deleted datapoint, @3%s@'; 4 'EvDpManager::cleanupDeletedDatapoint - default value config is deleted implicitly but still has overrides, @3%s@'; 5 'EvDpManager::cleanupDeletedDatapoint - initial value config is deleted implicitly for deleted datapoint, @3%s@'; 6 'EvDpManager::cleanupDeletedDatapoint - initial value config is deleted implicitly but still has overrides, @3%s@'; 7 'EvDpManager::cleanupDeletedDatapoint - distribution config is deleted implicitly for deleted datapoint, @3%s@'; 8 'EvDpManager::cleanupDeletedDatapoint - distribution config is deleted implicitly but still has overrides, @3%s@'; 9 'EvDpManager::cleanupDeletedDatapoint - rangeCheck config is deleted implicitly for deleted datapoint, @3%s@'; 10 'EvDpManager::cleanupDeletedDatapoint - rangeCheck config is deleted implicitly but still has overrides, @3%s@'

text list "SystemTextList_ConfigErrorAlarmTextLibrary_3": 1 'The configured data point type was deleted, but a configured type is still defined for the node type: @3%s@.'; 2 'The configured data point node type was deleted in the data point type, but a configured type is still defined for the element: @3%s@.'

text list "SystemTextList_ConfigErrorAlarmTextLibrary_4": 2 'Cycles: @6%s@ does not exist'; 3 'Alarms: @6%s@ exists already'; 4 'Tags: Address @6%s@ was rejected'; 1 'Connections: @6%s@ does not exist'; 5 'Tags: Acquisition mode @6%s@ is not supported.'; 6 'Cycles: @6%s@ was deleted but associated tags exist.'; 7 'Connections: @6%s@ was deleted but associated tags exist.'; 8 'Tags: Tag @6%s@ was rejected.'; 9 'Tags: Tag @6%s@ has an invalid value.'; 0 'Connections: Connection to @6%s@ could not be established.'; 65638 'Connections: Connection to @6%s@ could not be established.'; 65639 'Connections: @6%s@ disconnected.'; 65640 'Connections: Connection to the HMI device @6%s@ is lost.'; 65641 'Connections: Connection to the PLC @6%s@ is lost.'; 65541 'Connections: Timeout while establishing the connection to @6%s@.'; 65542 'Connections: @6%s@ faulty.'; 65543 'Connections: Connection to the HMI device disconnected. Connection @5%s@ was changed.'; 65544 'Connections: Connection to the HMI device disconnected. Driver property was changed for connection @5%s@.'

text list "SystemTextList_ConfigErrorAlarmTextLibrary_5": 1 'Connections: Lifecycle monitoring cycle must be shorter than the response time.'; 2 'Connections: Cyclic services are configured but not supported by the target device.'; 3 'Connections: Change-controlled reading is configured but not supported by the target device.'; 4 'Tags: The address @6%s@ does not exist in the PLC.'; 5 'Tags: The default conversion type for the address @6%s@ could not be determined.'; 6 'Tags: Invalid conversion type'; 7 'Cycles: Invalid conversion type. Conversion is not supported at HmiCycle.'; 4096 'Connections: Version of the address @6%s@ is not supported.'; 4097 'Connections: PROFIBUS address is not supported.'; 4098 'Connections: Softbus address is not supported.'; 4099 'Connections: Address type @6%s@ is not supported.'; 4100 'Connections: Invalid connection name @6%s@. Access point is being ignored.'; 4101 'Connections: Routing is not supported. @6%s@ is not used.'; 4102 'Connections: Routing is not supported. @6%s@ is not used.'; 4103 'Connections: Invalid IP address @6%s@'; 4104 'Connections: Invalid Named Connection @6%s@. Valid format: >VMD</>connection<'; 4105 'Connections: Invalid Named Connection @6%s@. VMD connection name is too long. Only 24 characters are permitted.'; 4106 'Connections: Invalid Named Connection @6%s@. Connection name is too long. Only 32 characters are permitted.'; 4107 'Connections: Rack number @6%s@ is outside of the permitted range (0..7)'; 4108 'Connections: Invalid Named Connection @6%s@. Rack is ignored.'; 4109 'Connections: Slot number @6%s@ is outside of the permitted range (0..31)'; 4110 'Connections: Invalid Named Connection @6%s@. Slot is ignored.'; 4111 'Connection could not be established. Maximum number of available connections (@6%s@) has been exceeded.'; 4112 'Connection aborted. No sign of life in the last @4%s@ ms.'; 4113 'Connection could not be established - @4%s@'; 4114 'Connection could not be established. The address @6%s@ cannot be used.'; 4115 'Connection could not be established. Invalid address @6%s@'; 4116 'Connection could not be established - @4%s@'

text list "SystemTextList_ConfigErrorAlarmTextLibrary_6": 1 'Connection could not be established. Application instance certificate is not configured.'; 2 'Connection could not be established. Server has rejected the client certificate. OPC UA status code @4%s@.'; 3 'Connection could not be established. Internal problem in the certificate store. OPC UA status code @4%s@'; 4 'Connection could not be established. Application instance certificate could not be loaded. OPC UA status code @4%s@'; 5 'Connection could not be established. Server has not provided a certificate. @4%s@'; 6 'Connection could not be established. Validation of server certificate has failed. OPC UA status code @4%s@.'; 7 'Connection was closed. Error during alarm synchronization. OPC UA status code @4%s@.'; 8 'Connection was closed. Alarm/event subscription has failed. The number of operations on the server has been exceeded.'; 9 'Connection was closed. Alarm/event subscription has failed. The number of alarm/event subscriptions on the server has been exceeded.'; 10 'Connection could not be established. Server reports a license problem. OPC UA status code @4%s@.'; 11 'Connection could not be established. Maximum number of server sessions has been exceeded.'; 12 'Connection could not be established. Safety configuration is inconsistent. @4%s@'; 13 'Connection could not be established. The address @4%s@ cannot be used.'; 14 'Connection could not be established. OPC UA status code @4%s@'; 15 'Connection aborted. OPC UA server was stopped.'; 16 'Connection aborted. No sign of life in the last @4%s@ ms.'; 17 'Connection was closed. OPC UA server maintenance.'; 18 'Connection could not be established. Invalid configuration of the authentication mode - @4%s@'; 19 'Connection could not be established. User could not be authenticated. OPC UA status code @4%s@'; 20 'Connection could not be established. Server does not permit anonymous connection. OPC UA status code @4%s@'; 21 'Connection could not be established. Certificate problem: Error when writing the safety-relevant data to @4%s@.'; 22 'Connection could not be established. Certificate problem: Unexpected file in the folder @4%s@ cannot be removed.'; 23 'Connection could not be established. User could not be authenticated. No user or password configured.'; 24 'Connection could not be established. Unexpected length of the server certificate. @4%s@'; 25 'Connection could not be established. @4%s@ is empty.'; 26 'Connection could not be established. @4%s@ has an unexpected format.'; 27 'Connection could not be established. Server endpoints cannot be read. OPC UA status code @4%s@'; 28 'Connection could not be established. No server endpoints were found. @4%s@'; 29 'Connection could not be established. Application instance certificate could not be found.'; 30 'Connection could not be established. Unexpected format of the certificate @4%s@.'; 31 'Connection could not be established. Unexpected format of the certificate block list @4%s@.'; 32 'Connection could not be established. User could not be authenticated. An encryption detail is invalid. @4%s@'; 34 'Connection could not be established. - The configured non-transparent redundancy mode @4%s@ is not supported.'; 101 'Tags: Address @6%s@ does not exist on the server.'; 103 'Tags: Address @6%s@ cannot be accessed.'; 104 'Tags: Acquisition mode is not supported for address @6%s@.'; 201 'Alarms: Address @6%s@ does not exist on the server.'; 202 'Alarms: Address @6%s@ cannot be used. The specified range filter is not an OPC UA Event Notifier.'; 203 'Alarms: Address @6%s@ cannot be used. The specified range filter does not exist on the server.'; 204 'Alarms: Address @6%s@ cannot be used because it is not an OPC UA event type.'; 205 'Alarms: Address @6%s@ cannot be used because the OPC UA condition type is not supported.'; 206 'Alarms: Address @6%s@ cannot be used because the event type does not exist on the server.'; 207 'Alarms: Acquisition type cannot be used for address @6%s@.'; 301 'Address @6%s@ cannot be used because the version number is missing.'; 302 'Address @6%s@ cannot be used because the version number is invalid.'; 303 'Address @6%s@ cannot be used because the number of '$' delimiters is invalid.'; 304 'Address @6%s@ cannot be used because the address type is invalid.'; 305 'Unsupported version @6%s@ of the address'; 401 'Unexpected OPC UA server response: @6%s@'

text list "SystemTextList_ConfigErrorAlarmTextLibrary_7": 1 'Messages: Invalid condition string for the alarm view @6%s@.'; 2 'Messages: Invalid status tag and bit for the alarm view @6%s@.'; 3 'Messages: Invalid control tag and bit for the alarm view @6%s@.'

text list "SystemTextList_ConfigErrorAlarmTextLibrary_8": 1 'Logs: Implicit deletion. Logging tag instance @6%s@ should be deleted but there are overloaded elements.'

text list "SystemTextList_ConfigErrorAlarmTextLibrary_9": 2 'Restart of the runtime is required.'; 3 'The correct storage medium must be ejected and inserted again.'

text list "SystemTextList_ConfigErrorAlarmTextLibrary_10": 1 'CDS cache - Cache folder cannot be created or reached: @6%s@'; 2 'LOC cache - Cache folder cannot be created or reached: @6%s@'

text list "SystemTextList_ConfigErrorAlarmTextLibrary_11": 2 'and synchronization will start automatically. Shutting down either of them during synchronization will not cause data loss.'; 3 'and synchronization is scheduled for: @5%Y-%m-%d %H:%M:%S@. Shutting down either of the computers will not cause data loss.'

text list "SystemTextList_RuntimeCollaborationFailureReason_1": 0 'Unknown error (@3%s@)'; 1 'The system is not running or there is a network problem'; 2 'Runtime is not started on the target device.'; 3 'The System ID does not match the expected System ID (@3%s@)'; 4 'The Collaboration name does not match the expected Collaboration name '@3%s@''; 5 'Wrong or unknown certificate'; 6 'Revoked certificate'; 7 'The time difference is too big.'; 8 'No common supported message version'; 9 'System ID (@3%s@) already exists'; 10 'System name (@3%s@) already exists'; 11 'ID/Name in local configuration for Runtime Collaboration already exists'

text list "SystemTextList_RedundancyRecoveryFailureReason_1": 0 'Data recovery request temporarily rejected until own recovery request has been responded to.'; 1 'Data recovery request rejected. Online backup running.'; 2 'Data recovery request rejected. Connection to the Event Manager is not established.'; 3 'Data recovery request temporarily rejected until delta activation is complete.'; 4 'Data recovery request temporarily rejected until alarms and tags are retentive.'; 5 'Data recovery request rejected. The obligatory file config.level.es is missing on the computer.'; 6 'Data recovery request was canceled by the Event Manager.'; 7 'The data synchronization between the devices has failed.'

text list "SystemTextList_S7PlusAlarmTextListCollection_1": 4096 'Connections: Connection to the PLC @4%s@ is lost'; 4097 'Connections: Connection to the HMI device @4%s@ is lost'; 4098 'Connections: Maximum number of connections exceeded - @4%s@'; 4099 'Out of resources on PLC - @4%s@'; 4100 'Legitimation failed, invalid or missing password - @4%s@'; 4101 'Request to open the connection failed - @4%s@'; 4102 'Connections: Cannot connect to PLC - @4%s@'; 4103 'Request to open the connection could not be sent'; 4104 'General certificate error for PLC - @4%s@'; 4105 'PLC certificate expired for PLC - @4%s@'; 4106 'PLC certificate is revoked for PLC - @4%s@'; 4107 'PLC certificate is untrustworthy. Manual trust is possible for - @4%s@'; 4108 'PLC certificate is untrustworthy. Manual trust is not possible for - @4%s@'

text list "SystemTextList_AllenBradleyEIPAlarmTextListCollection_7": 4096 'Connection lost on PLC side - @5%s@'; 4097 'Connection lost on HMI side - @5%s@'; 4098 'Maximum number of connections exceeded - @5%s@'; 4099 'Out of resources on PLC - @5%s@'; 4100 'Legitimation failed, invalid or missing password - @5%s@'; 4101 'Open request failed - @5%s@'; 4102 'Cannot connect to PLC - @5%s@'; 4103 'Open request could not be sent'; 4104 'root certificate expired for - @5%s@'; 4105 'PLC certificate untrusted for - @5%s@'

text list "SystemTextList_AllenBradleyDF1AlarmTextListCollection_9": 4096 'Connections: Connection to the PLC @5%s@ is lost'; 4097 'Connections: Connection to the HMI device @5%s@ is lost'; 4098 'Connections: Maximum number of connections exceeded - @5%s@'; 4099 'Out of resources on PLC - @5%s@'; 4100 'Legitimation failed, invalid or missing password - @5%s@'; 4101 'Request to open the connection failed - @5%s@'; 4102 'Connections: Cannot connect to PLC - @5%s@'; 4103 'Request to open the connection could not be sent'; 4104 'General certificate error for PLC - @5%s@'; 4105 'PLC certificate expired for PLC - @5%s@'; 4106 'PLC certificate is revoked for PLC - @5%s@'; 4107 'PLC certificate is untrustworthy. Manual trust is possible for - @5%s@'; 4108 'PLC certificate is untrustworthy. Manual trust is not possible for - @5%s@'

text list "SystemTextList_OmronEIPAlarmTextListCollection_6": 4096 'Connection lost on PLC side - @5%s@'; 4097 'Connection lost on HMI side - @5%s@'; 4098 'Maximum number of connections exceeded - @5%s@'; 4099 'Out of resources on PLC - @5%s@'; 4100 'Legitimation failed, invalid or missing password - @5%s@'; 4101 'Open request failed - @5%s@'; 4102 'Cannot connect to PLC - @5%s@'; 4103 'Open request could not be sent'; 4104 'root certificate expired for - @5%s@'; 4105 'PLC certificate untrusted for - @5%s@'

text list "SystemTextList_StdModbusTCPAlarmTextListCollection_5": 4096 'Connections: Connection to the PLC @5%s@ is lost'; 4097 'Connections: Connection to the HMI device @5%s@ is lost'; 4098 'Connections: Maximum number of connections exceeded - @5%s@'; 4099 'Out of resources on PLC - @5%s@'; 4100 'Legitimation failed, invalid or missing password - @5%s@'; 4101 'Request to open the connection failed - @5%s@'; 4102 'Connections: Cannot connect to PLC - @5%s@'; 4103 'Request to open the connection could not be sent'; 4104 'General certificate error for PLC - @5%s@'; 4105 'PLC certificate expired for PLC - @5%s@'; 4106 'PLC certificate is revoked for PLC - @5%s@'; 4107 'PLC certificate is untrustworthy. Manual trust is possible for - @5%s@'; 4108 'PLC certificate is untrustworthy. Manual trust is not possible for - @5%s@'

text list "SystemTextList_MitsubishiMCAlarmTextListCollection_4": 4096 'Connection lost on PLC side - @5%s@'; 4097 'Connection lost on HMI side - @5%s@'; 4098 'Maximum number of connections exceeded - @5%s@'; 4099 'Out of resources on PLC - @5%s@'; 4100 'Legitimation failed, invalid or missing password - @5%s@'; 4101 'Open request failed - @5%s@'; 4102 'Cannot connect to PLC - @5%s@'; 4103 'Open request could not be sent'; 4104 'root certificate expired for - @5%s@'; 4105 'PLC certificate untrusted for - @5%s@'

text list "SystemTextList_MitsubishiiQAlarmTextListCollection_3": 4096 'Connection lost on PLC side - @5%s@'; 4097 'Connection lost on HMI side - @5%s@'; 4098 'Maximum number of connections exceeded - @5%s@'; 4099 'Out of resources on PLC - @5%s@'; 4100 'Legitimation failed, invalid or missing password - @5%s@'; 4101 'Open request failed - @5%s@'; 4102 'Cannot connect to PLC - @5%s@'; 4103 'Open request could not be sent'; 4104 'root certificate expired for - @5%s@'; 4105 'PLC certificate untrusted for - @5%s@'

text list "SystemTextList_StdModbusRTUAlarmTextListCollection_8": 4096 'Connections: Connection to the PLC @5%s@ is lost'; 4097 'Connections: Connection to the HMI device @5%s@ is lost'; 4098 'Connections: Maximum number of connections exceeded - @5%s@'; 4099 'Out of resources on PLC - @5%s@'; 4100 'Legitimation failed, invalid or missing password - @5%s@'; 4101 'Request to open the connection failed - @5%s@'; 4102 'Connections: Cannot connect to PLC - @5%s@'; 4103 'Request to open the connection could not be sent'; 4104 'General certificate error for PLC - @5%s@'; 4105 'PLC certificate expired for PLC - @5%s@'; 4106 'PLC certificate is revoked for PLC - @5%s@'; 4107 'PLC certificate is untrustworthy. Manual trust is possible for - @5%s@'; 4108 'PLC certificate is untrustworthy. Manual trust is not possible for - @5%s@'

text list "SystemTextList_LogoAlarmTextListCollection_10": 4096 'Connections: Connection to the PLC @5%s@ is lost'; 4097 'Connections: Connection to the HMI device @5%s@ is lost'; 4098 'Connections: Maximum number of connections exceeded - @5%s@'; 4099 'Out of resources on PLC - @5%s@'; 4100 'Legitimation failed, invalid or missing password - @5%s@'; 4101 'Request to open the connection failed - @5%s@'; 4102 'Connections: Cannot connect to PLC - @5%s@'; 4103 'Request to open the connection could not be sent'; 4104 'General certificate error for PLC - @5%s@'; 4105 'PLC certificate expired for PLC - @5%s@'; 4106 'PLC certificate is revoked for PLC - @5%s@'; 4107 'PLC certificate is untrustworthy. Manual trust is possible for - @5%s@'; 4108 'PLC certificate is untrustworthy. Manual trust is not possible for - @5%s@'
*)